FUNCTION HLI_ChannelGetMode : DWORD
VAR_INPUT
	nChan					: UDINT;			(* Number of channel *)
END_VAR
VAR
	nHliChIdx			: UDINT;
END_VAR

(* ========================================================= *)
(*    FUN: HLI_ChannelGetMode                                *)
(* --------------------------------------------------------- *)
(*   Desc:                                                   *)
(* Author: MK                                                *)
(*   Date: 21.12.2011                                        *)
(*   Rev.: 1.0                                               *)
(* ========================================================= *)


nHliChIdx := nChan - 1;

IF nChan <= 0 OR gNrCh < nChan OR			(* check for channel no *)
	gpCh[nHliChIdx] = 0 THEN					(* check for zero pointer *)
	HLI_ChannelGetMode := 0;
	RETURN; (* e x i t *)
END_IF

(* if the stop button from the HMI is selected the request is set *)
HLI_ChannelGetMode := gpCh[nHliChIdx]^.channel_mc_control.mode_and_state.state_r.mode;

END_FUNCTION

(* stored: Version 1.1.0.1, ProductVersion 3.1.4018.5
   POU HLI_ChannelGetMode: Id {6e420aed-172e-4934-ab1f-e7aad7bfc266}, SpecialFunc None *)
